Universal Robots PolyScope program: 8Ds.urp

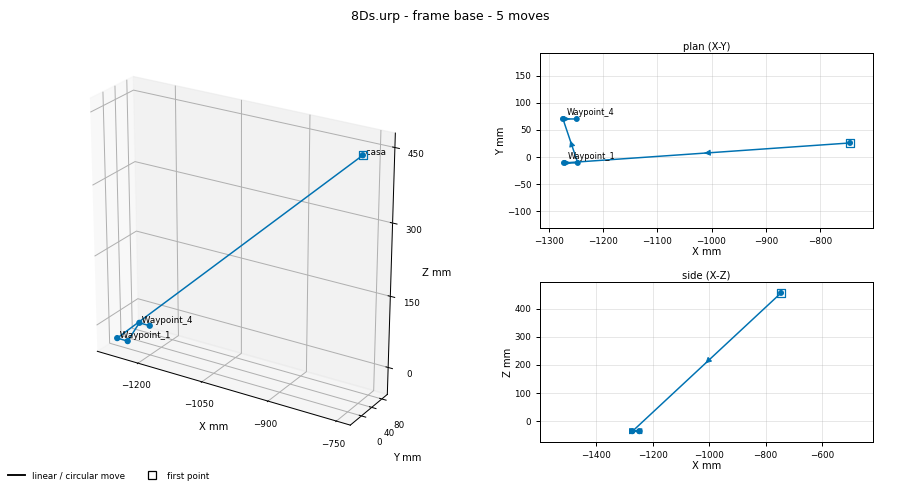
[picture p0: tool path of 8Ds.urp in frame base, 5 of 6 moves have a stored position in this frame; points joined in program order, loops and branches not executed]
Program 8Ds (installation=instalacion_derecha_10_MAR_21 directory=/programs/8Ds createdIn=5.6.0.90886 lastSavedIn=5.6.0.90886 robotSerialNumber=20195001785)
Calibrated DH parameters: a=[0.000107, -0.568984, -0.552934, -0.00001, -0.000063, 0]; d=[0.180718, -257.998067, 200.685024, 57.48776, 0.119923, 0.115353]; alpha=[1.571119, 0.000876, -0.002498, 1.571178, -1.570523, 0]; deltaTheta=[0, -0.378191, 0.631587, -0.253396, 0, 0]
Robot Program (runOnlyOnce=false)
  MoveL speed 250 mm/s, acceleration 1200 mm/s^2 (useActiveTCP=true) feature=Base
    alpha := 6
    Loop Forever
      SuppressedNode
        Waypoint Waypoint_3: TCP in base x=-133.824 y=-733.308 z=19.085 mm, rx=3.0039 ry=-0.8902 rz=-0.004 rad; joints [66.097, -73.504, 119.465, -45.965, 89.924, 0.082] deg; TCP offset x=0.411 y=-218.298 z=37.994 mm, rx=1.558 ry=-0.1255 rz=0.1212 rad
      Waypoint casa: TCP in base x=-744.966 y=25.975 z=455.169 mm, rx=1.6931 ry=-2.6406 rz=-0.0118 rad; joints [-15.574, -90.004, 90.001, 0, 90, 0] deg; TCP offset x=0.411 y=-218.298 z=37.994 mm, rx=1.558 ry=-0.1255 rz=0.1212 rad
      Waypoint Waypoint_1: TCP in base x=-1271.558 y=-10.798 z=-35 mm, rx=1.6931 ry=-2.6407 rz=-0.0118 rad; joints [-6.287, -24.768, 38.356, -13.597, 99.266, 0.063] deg; TCP offset x=0.411 y=-218.298 z=37.994 mm, rx=1.558 ry=-0.1255 rz=0.1212 rad
      Waypoint Waypoint_2: TCP in base x=-1246.186 y=-10.793 z=-35 mm, rx=1.6931 ry=-2.6406 rz=-0.0118 rad; joints [-6.432, -28.248, 45.296, -17.06, 99.108, 0.066] deg
      Waypoint Waypoint_4: TCP in base x=-1273.448 y=70.144 z=-35 mm, rx=1.6931 ry=-2.6407 rz=-0.0118 rad; joints [-10.4, -24.603, 38.025, -13.428, 95.153, 0.063] deg; TCP offset x=0.411 y=-218.298 z=37.994 mm, rx=1.558 ry=-0.1255 rz=0.1212 rad
      Waypoint Waypoint_5: TCP in base x=-1248.05 y=70.124 z=-34.981 mm, rx=1.6931 ry=-2.6406 rz=-0.0118 rad; joints [-10.639, -28.11, 45.021, -16.916, 94.904, 0.065] deg
      Loop Counting (count=10) loopVariable(name=Loop_2)
        internos := interpolate_pose(Waypoint_4, Waypoint_5, alpha)
        Waypoint Waypoint (Variable): variable=internos
        MoveDirectionNode (selectedDirection=ZMinus toolParams=0.0015, 0.005)
          Until TOOL_CONTACT_DETECTION (allowActions=false retraction=0 decelerationAcceleration=9 decelerationAngularAcceleration=34.906585)
        Wait Sleep waitTime=1
        Popup Message (haltProgram=false message=kokl inputType=Text)
        MoveDirectionNode (selectedDirection=ZPlus)
          Until DISTANCE (allowActions=false deceleration=3 distanceNodeType=STOP) Distance=0.05; motionParameters(blendRadius=0)
        alpha := alpha+1
